FUNCTION_BLOCK Test_AggregateResult_Busy EXTENDS T_UnitTestBase
VAR
	ResultAggregate : T_ResultAggregate;
	Execution1 : T_Execution;
	Execution2 : T_Execution;
	Execution3 : T_Execution;
END_VAR

METHOD Init
SUPER^.Init();

Execution1.FB_init(FALSE,FALSE);
Execution2.FB_init(FALSE,FALSE);
Execution3.FB_init(FALSE,FALSE);
END_METHOD

{attribute 'analysis' := '-33'} // inhibit unused variable warning
METHOD RunTest
ResultAggregate.ClearResults();

ResultAggregate.AddResult(Execution1);
ResultAggregate.AddResult(Execution2);
ResultAggregate.AddResult(Execution3);

AssertIsTrue(Condition := ResultAggregate.Busy = FALSE,
             Message   := 'ResultAggregate.Busy is not false');

Execution1.Start();
Execution1.SetBusy();

AssertIsTrue(Condition := ResultAggregate.Busy = TRUE,
             Message   := 'ResultAggregate.Busy is false');

TestCompleted := TRUE;
END_METHOD

END_FUNCTION_BLOCK

(* stored: Version 1.1.0.1, ProductVersion 3.1.4024.12
   POU Test_AggregateResult_Busy: Id {5ee0aa7d-00d6-433e-bb66-fb3816002789}, SpecialFunc None
   Method Init: Id {10d5e106-bf7a-4578-ba85-5cbfd17c8f16}
   Method RunTest: Id {d2211e7e-8e5d-47ef-9b39-832160780443} *)
